FUNCTION_BLOCK Matstation
  (* Version 0.1, 2005-04-08, JohanPetter, Chalmers *)
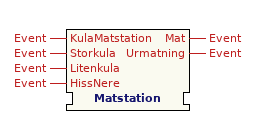
  EVENT_INPUT
    KulaMatstation;
    Storkula;
    Litenkula;
    HissNere;
  END_EVENT
  EVENT_OUTPUT
    Mat;
    Urmatning;
  END_EVENT
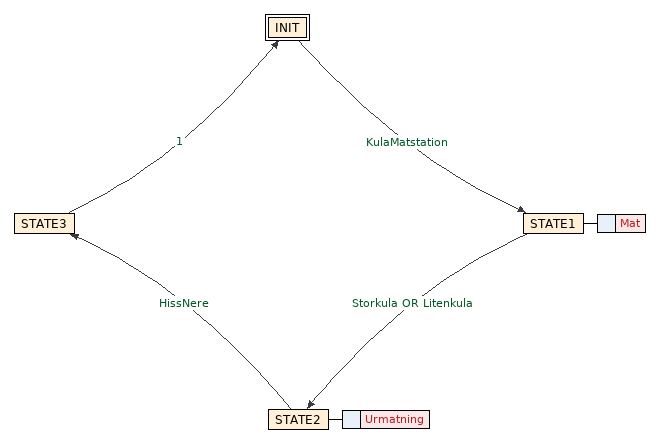
  EC_STATES
    INIT;
    STATE1 : -> Mat;
    STATE2 : -> Urmatning;
    STATE3;
  END_STATES
  EC_TRANSITIONS
    INIT TO STATE1 := KulaMatstation;
    STATE1 TO STATE2 := Storkula OR Litenkula;
    STATE2 TO STATE3 := HissNere;
    STATE3 TO INIT := 1;
  END_TRANSITIONS
END_FUNCTION_BLOCK
